FUNCTION_BLOCK FB_EventHandler
VAR_INPUT
	bExecute	: BOOL;
	eEventName	: E_Events;
	sSystem		: STRING;
	sMessage	: STRING;
END_VAR

VAR_OUTPUT
	bDone		: BOOL := FALSE;
END_VAR

VAR
	fbMessage	: FB_TcMessage;
	bSend 		: BOOL := FALSE;
END_VAR

// Raising the events for each event class
CASE eEventName OF 

	E_Events.INFO: //INFO Event
		IF bExecute THEN
			bExecute := FALSE;
			fbMessage.CreateEx(TC_EVENTS.ASRS.Info, 0);
			fbMessage.ipArguments.AddString(sSystem).AddString(sMessage);
			bSend	:= TRUE;
		END_IF
	
	E_Events.WARNING: //Warning Event
		IF bExecute THEN
				bExecute := FALSE;
				fbMessage.CreateEx(TC_EVENTS.ASRS.Warning, 0);
				fbMessage.ipArguments.AddString(sSystem).AddString(sMessage);
				bSend	:= TRUE;
			END_IF
			
	E_Events.ERROR: //Error Event
		IF bExecute THEN
			bExecute := FALSE;
			fbMessage.CreateEx(TC_EVENTS.ASRS.Error, 0);
			fbMessage.ipArguments.AddString(sSystem).AddString(sMessage);
			bSend	:= TRUE;
		END_IF
	
	E_Events.CRITICAL: //Critical Event
		IF bExecute THEN
			bExecute := FALSE;
			fbMessage.CreateEx(TC_EVENTS.ASRS.Critical, 0);
			fbMessage.ipArguments.AddString(sSystem).AddString(sMessage);
			bSend	:= TRUE;
		END_IF
	
END_CASE

//Sending the event message
IF bSend THEN
	fbMessage.Send(0);
	bDone := TRUE;
	bSend := FALSE;
END_IF

END_FUNCTION_BLOCK

(* stored: Version 1.1.0.1, ProductVersion 3.1.4024.12
   POU FB_EventHandler: Id {50d7dbe2-9dbf-4c79-9105-c09bc47664b0}, SpecialFunc None *)
